FUNCTION_BLOCK AllNextFeedDone (* Basic Function Block Type *)
  (* Standard: 61499-2 *)
  (* Version 0.0, 7/16/2026, Schneider Electric, Template *)
  PACKAGE SE.Nereda;
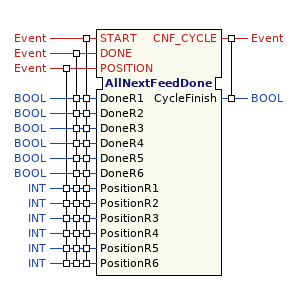
  EVENT_INPUT
    START WITH DoneR1, DoneR2, DoneR3, DoneR4, DoneR5, DoneR6, PositionR1, PositionR2, PositionR3, PositionR4, PositionR5, PositionR6;
    DONE WITH DoneR1, DoneR2, DoneR3, DoneR4, DoneR5, DoneR6, PositionR1, PositionR2, PositionR3, PositionR4, PositionR5, PositionR6; (* Normal Execution Request *)
    POSITION WITH PositionR1, PositionR2, PositionR3, PositionR4, PositionR5, PositionR6;
  END_EVENT
  EVENT_OUTPUT
    CNF_CYCLE WITH CycleFinish; (* Execution Confirmation *)
  END_EVENT
  VAR_INPUT
    DoneR1 : BOOL;
    DoneR2 : BOOL;
    DoneR3 : BOOL;
    DoneR4 : BOOL;
    DoneR5 : BOOL;
    DoneR6 : BOOL;
    PositionR1 : INT;
    PositionR2 : INT;
    PositionR3 : INT;
    PositionR4 : INT;
    PositionR5 : INT;
    PositionR6 : INT;
  END_VAR
  VAR_OUTPUT
    CycleFinish : BOOL;
  END_VAR
  VAR
    InDoneR1 : BOOL;
    InDoneR2 : BOOL;
    InDoneR3 : BOOL;
    InDoneR4 : BOOL;
    InDoneR5 : BOOL;
    InDoneR6 : BOOL;
  END_VAR
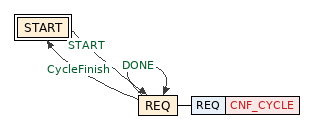
  EC_STATES
    START; (* Initial State *)
    REQ : REQ -> CNF_CYCLE;
  END_STATES
  EC_TRANSITIONS
    START TO REQ := START;
    REQ TO START := CycleFinish;
    REQ TO REQ := DONE;
  END_TRANSITIONS
  ALGORITHM REQ IN ST: (* Normally executed algorithm *)
;
IF PositionR1 > 0 THEN
	InDoneR1 := DoneR1;
ELSE
	InDoneR1 := TRUE;
END_IF;

IF PositionR2 > 0 THEN
	InDoneR2 := DoneR2;
ELSE
	InDoneR2 := TRUE;
END_IF;

IF PositionR3 > 0 THEN
	InDoneR3 := DoneR3;
ELSE
	InDoneR3 := TRUE;
END_IF;

IF PositionR4 > 0 THEN
	InDoneR4 := DoneR4;
ELSE
	InDoneR4 := TRUE;
END_IF;

IF PositionR5 > 0 THEN
	InDoneR5 := DoneR5;
ELSE
	InDoneR5 := TRUE;
END_IF;

IF PositionR6 > 0 THEN
	InDoneR6 := DoneR6;
ELSE
	InDoneR6 := TRUE;
END_IF;

CycleFinish := InDoneR1 AND InDoneR2 AND InDoneR3 AND InDoneR4 AND InDoneR5 AND InDoneR6;
  END_ALGORITHM
END_FUNCTION_BLOCK
